// TIA Portal V21 export
FUNCTION_BLOCK "EdgeParts"   // FB42, LAD
   VAR_TEMP   // added for the SCL form of the ladder/FBD networks
      _w1 : Bool;
   END_VAR
BEGIN

REGION Network 1: PContact
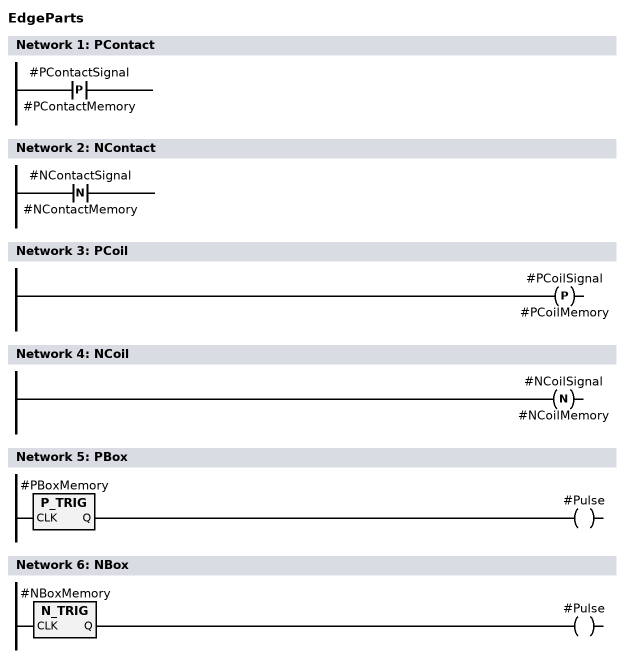
   #_w1 := #PContactSignal AND NOT #PContactMemory;   // rising edge of #PContactSignal
   #PContactMemory := #PContactSignal;
END_REGION

REGION Network 2: NContact
   #_w1 := NOT #NContactSignal AND #NContactMemory;   // falling edge of #NContactSignal
   #NContactMemory := #NContactSignal;
END_REGION

REGION Network 3: PCoil
   #PCoilSignal := NOT #PCoilMemory;   // rising edge
   #PCoilMemory := TRUE;
END_REGION

REGION Network 4: NCoil
   #NCoilSignal := NOT TRUE AND #NCoilMemory;   // falling edge
   #NCoilMemory := TRUE;
END_REGION

REGION Network 5: PBox
   RUNG wire#powerrail
      P_Trig( #PBoxMemory )
      Coil( #Pulse )
   END_RUNG
   // the same network as SCL:
   #_w1 := NOT #PBoxMemory;   // rising edge
   #PBoxMemory := TRUE;
   #Pulse := #_w1;
END_REGION

REGION Network 6: NBox
   RUNG wire#powerrail
      N_Trig( #NBoxMemory )
      Coil( #Pulse )
   END_RUNG
   // the same network as SCL:
   #_w1 := NOT TRUE AND #NBoxMemory;   // falling edge
   #NBoxMemory := TRUE;
   #Pulse := #_w1;
END_REGION
END_FUNCTION_BLOCK
